FUNCTION_BLOCK TransportSequenceStop EXTENDS TransportSequence IMPLEMENTS ZCore.ISequence
VAR
  _step : ZCore.Step(TransportStep.StopBegin, TransportStep.StopEnd);
  _timerSim : ZAux.Timer;
END_VAR

IF OnStart(_step) THEN
  ; // init custom sequence variables here ...
END_IF

REPEAT
  LogStep();

  CASE _step.Index OF
    (* -------------------------------------------------------------------------------------------------------------------------------- *)
    TransportStep.StopBegin:
    (* -------------------------------------------------------------------------------------------------------------------------------- *)
      IF _step.OnEntry()
      THEN
        _axis.HorizontalX.StopAsync(startToken:=THIS^);
        _axis.VerticalZ.StopAsync(startToken:=THIS^);
			END_IF
      
      Await2(obj1:=_axis.HorizontalX, obj2:=_axis.VerticalZ, nextStep:=TransportStep.StopEnd);

    (* -------------------------------------------------------------------------------------------------------------------------------- *)
    TransportStep.StopEnd:
    (* -------------------------------------------------------------------------------------------------------------------------------- *)    
      SetBusy(FALSE);
  
  ELSE
    Abort('sequence contains unhandled step');
  END_CASE
UNTIL _step.IsNotRepeatable() OR_ELSE NOT Busy END_REPEAT

END_FUNCTION_BLOCK

(* stored: Version 1.1.0.1
   POU TransportSequenceStop: Id {d9c682e7-474a-4a1c-8c3c-18fa003de899}, SpecialFunc None *)
